(* PLC project Generated.project, CODESYS CODESYS V3.5 SP19 Patch 1 *)
(* stored: creationDateTime 2026-11-16T13:11:40.466311, modificationDateTime 2026-11-16T13:11:40.466311 *)

(* DOC: DOC/AF/AF_Partie-13_Fonction_Simulation_v2.5.md Capteur de position cumulatif avec hysteresis et episode intermittent rejouable. Cette brique ne connait ni le mouvement ni la logique M3 : elle transforme uniquement une position mecanique vraie en DI. *)
FUNCTION_BLOCK FB_Sim_PositionSensor
  VAR_INPUT
    Enable : BOOL;
    Position_M : REAL;
    Threshold_M : REAL;
    Hysteresis_M : REAL := 0.02;
    ActiveBelowThreshold : BOOL := TRUE;
    ElectricalDelayS : REAL := 0;
    IntermittenceActive : BOOL := FALSE;
    IntermittenceDurationS : REAL := 1;
    IntermittencePeriodS : REAL := 0.12;
    ScenarioSeed : UDINT := 1;
    CycleTimeS : REAL := 0.01;
    BlipTransitions : UDINT := 0;  (* Profil « BLIP COURT » — SECOND profil, independant du train de bascules du profil d'intermittence ci-dessus (dont les parametres restent inchanges). 0 = desactive : le comportement historique est strictement conserve. Rejoue les excursions electriques courtes mesurees sur la trace terrain du 2026-09-04 : Tremie contradictoire pendant 2 echantillons a 12,24 s (~200 ms) et PV reactive 1 echantillon a 14,94 s (~100 ms). BlipTransitions = nombre de bascules electriques (1 = une excursion puis retour) ; BlipDurationS = duree de maintien de chaque etat, donc largeur de l'excursion. *)
    BlipDurationS : REAL := 0.2;
    CamDropoutActive : BOOL := FALSE;  (* L5 (2026-10-28) — MECANISME DE CAME, SPATIAL : en franchissant le capteur on le VOIT, on le PERD sur une courte zone, on le RETROUVE, puis il reste FIXE. Lie a la POSITION (pas au temps) : se produit a chaque passage, dans les DEUX sens, et reste stable a l'arret (bornes de la zone avec hysteresis CST_CamHysteresis_M contre le bruit/balancement). Zone de perte placee APRES le front de detection (cote -/+ Hysteresis_M) : [front - Start - Width ; front - Start] cote detection. FALSE = historique strictement inchange. Valeurs = HYPOTHESES. *)
    CamDropoutStart_M : REAL := 0.02;
    CamDropoutWidth_M : REAL := 0.04;
    FiniteCamActive : BOOL := FALSE;  (* Came finie : FALSE = capteur cumulatif ; TRUE = sortie active uniquement sur CamLength_M apres Threshold_M. *)
    CamLength_M : REAL := 0;
  END_VAR
  VAR_OUTPUT
    RawDetected : BOOL;
    ElectricalOutput : BOOL;
    EpisodeActive : BOOL;
    BlipActive : BOOL;
    TransitionCount : UDINT;
    EpisodeTogglePeriodS : REAL;
  END_VAR
  VAR
    Initialized : BOOL;
    PreviousRawDetected : BOOL;
    EpisodeTarget : BOOL;
    DelayTimerS : REAL;
    EpisodeTimerS : REAL;
    ToggleTimerS : REAL;
    RandomState : UDINT;
    BlipRunning : BOOL;
    BlipTimerS : REAL;
    BlipCount : UDINT;
    HystDetected : BOOL;  (* L5 : etat mecanique avec hysteresis (avant perte de came) *)
    InCamDropout : BOOL;  (* L5 : position dans la zone de perte de la came *)
    CamNear_M : REAL;  (* L5 : borne de la zone cote front de detection *)
    CamFar_M : REAL;  (* L5 : borne de la zone cote interieur *)
    PastFiniteCam : BOOL;  (* Depassement au-dela de la longueur physique de came *)
    CamEnd_M : REAL;  (* Borne de fin de came finie *)
    CST_BlipMaxTransitions : UDINT := 1000;  (* Plafond du nombre de bascules du profil « blip court » : borne la duree de l'episode et interdit tout rebouclage de compteur UDINT (revue du 2026-09-20, F9). *)
    CST_CamHysteresis_M : REAL := 0.01;  (* L5 : hysteresis des bornes de la zone de perte *)
  END_VAR

            

IF NOT Enable THEN
    Initialized := FALSE;
    RawDetected := FALSE;
    ElectricalOutput := FALSE;
    PreviousRawDetected := FALSE;
    EpisodeActive := FALSE;
    BlipActive := FALSE;
    BlipRunning := FALSE;
    BlipTimerS := 0.0;
    BlipCount := 0;
    DelayTimerS := 0.0;
    EpisodeTimerS := 0.0;
    ToggleTimerS := 0.0;
    TransitionCount := 0;
    EpisodeTogglePeriodS := 0.0;
    PastFiniteCam := FALSE;
    RETURN;
END_IF;

(* Hysteresis sur une frontiere cumulative : les cinq DI restent compatibles avec
   le mot thermometre du decodeur M3, contrairement a cinq fenetres independantes. *)
IF NOT Initialized THEN
    IF ActiveBelowThreshold THEN
        RawDetected := Position_M <= Threshold_M;
        IF FiniteCamActive THEN
            PastFiniteCam := Position_M < (Threshold_M - MAX(0.0, CamLength_M));
            RawDetected := RawDetected AND NOT PastFiniteCam;
        ELSE
            PastFiniteCam := FALSE;
        END_IF;
    ELSE
        RawDetected := Position_M >= Threshold_M;
        IF FiniteCamActive THEN
            PastFiniteCam := Position_M > (Threshold_M + MAX(0.0, CamLength_M));
            RawDetected := RawDetected AND NOT PastFiniteCam;
        ELSE
            PastFiniteCam := FALSE;
        END_IF;
    END_IF;
    HystDetected := RawDetected;
    ElectricalOutput := RawDetected;
    PreviousRawDetected := RawDetected;
    RandomState := ScenarioSeed MOD 1000000;
    IF RandomState = 0 THEN
        RandomState := 1;
    END_IF;
    EpisodeTogglePeriodS := MAX(0.01, IntermittencePeriodS);
    Initialized := TRUE;
    RETURN;
END_IF;

IF ActiveBelowThreshold THEN
    IF HystDetected THEN
        HystDetected := Position_M <= (Threshold_M + MAX(0.0, Hysteresis_M));
    ELSE
        HystDetected := Position_M <= (Threshold_M - MAX(0.0, Hysteresis_M));
    END_IF;
    (* Zone de perte : apres le front d'entree en detection (cote - hysteresis), vers l'interieur. *)
    CamNear_M := Threshold_M - MAX(0.0, Hysteresis_M) - MAX(0.0, CamDropoutStart_M);
    CamFar_M := CamNear_M - MAX(0.0, CamDropoutWidth_M);
    IF NOT CamDropoutActive THEN
        InCamDropout := FALSE;
    ELSIF InCamDropout THEN
        InCamDropout := (Position_M <= CamNear_M + CST_CamHysteresis_M) AND (Position_M > CamFar_M - CST_CamHysteresis_M);
    ELSE
        InCamDropout := (Position_M <= CamNear_M - CST_CamHysteresis_M) AND (Position_M > CamFar_M + CST_CamHysteresis_M);
    END_IF;
    CamEnd_M := Threshold_M - MAX(0.0, CamLength_M);
    IF NOT FiniteCamActive THEN
        PastFiniteCam := FALSE;
    ELSIF PastFiniteCam THEN
        PastFiniteCam := Position_M < (CamEnd_M + CST_CamHysteresis_M);
    ELSE
        PastFiniteCam := Position_M < CamEnd_M;
    END_IF;
ELSE
    IF HystDetected THEN
        HystDetected := Position_M >= (Threshold_M - MAX(0.0, Hysteresis_M));
    ELSE
        HystDetected := Position_M >= (Threshold_M + MAX(0.0, Hysteresis_M));
    END_IF;
    CamNear_M := Threshold_M + MAX(0.0, Hysteresis_M) + MAX(0.0, CamDropoutStart_M);
    CamFar_M := CamNear_M + MAX(0.0, CamDropoutWidth_M);
    IF NOT CamDropoutActive THEN
        InCamDropout := FALSE;
    ELSIF InCamDropout THEN
        InCamDropout := (Position_M >= CamNear_M - CST_CamHysteresis_M) AND (Position_M < CamFar_M + CST_CamHysteresis_M);
    ELSE
        InCamDropout := (Position_M >= CamNear_M + CST_CamHysteresis_M) AND (Position_M < CamFar_M - CST_CamHysteresis_M);
    END_IF;
    CamEnd_M := Threshold_M + MAX(0.0, CamLength_M);
    IF NOT FiniteCamActive THEN
        PastFiniteCam := FALSE;
    ELSIF PastFiniteCam THEN
        PastFiniteCam := Position_M > (CamEnd_M - CST_CamHysteresis_M);
    ELSE
        PastFiniteCam := Position_M > CamEnd_M;
    END_IF;
END_IF;
(* L5 : perte de came + came finie ; hors options, RawDetected = HystDetected. *)
RawDetected := HystDetected AND NOT InCamDropout AND NOT PastFiniteCam;

(* Un episode est declenche par un franchissement mecanique, pas par une de ses
   propres bascules electriques. Les fronts restent donc bornes et reproductibles. *)
IF RawDetected <> PreviousRawDetected THEN
    PreviousRawDetected := RawDetected;
    EpisodeTarget := RawDetected;
    (* Une bascule mecanique pendant l'episode modifie seulement la cible finale.
       Elle ne remet jamais son chronometre a zero : l'episode reste borne. *)
    IF NOT EpisodeActive THEN
        DelayTimerS := 0.0;
        EpisodeTimerS := 0.0;
        ToggleTimerS := 0.0;
        (* Tirage unique par episode : reproductible pour une graine et sans bruit
           blanc scan-par-scan. La periode varie de 70 % a 130 % du nominal. *)
        RandomState := RandomState + 7919;
        IF RandomState >= 1000000 THEN
            RandomState := RandomState - 1000000;
        END_IF;
        EpisodeTogglePeriodS := MAX(0.01, IntermittencePeriodS
            * (0.7 + UDINT_TO_REAL(RandomState MOD 6000) / 10000.0));
        EpisodeActive := IntermittenceActive AND (IntermittenceDurationS > 0.0);
    END_IF;
    (* Blip court : arme sur le meme front MECANIQUE. Ses propres bascules electriques ne
       peuvent donc jamais le rearmer — meme protection que l'episode d'intermittence. *)
    IF (BlipTransitions > 0) AND (BlipDurationS > 0.0) THEN
        BlipRunning := TRUE;
        BlipTimerS := 0.0;
        BlipCount := 0;
        BlipActive := TRUE;
        (* Ecretage : au-dela de ce plafond, un compteur UDINT pourrait reboucler et rendre
           le blip non terminant (revue du 2026-09-20, F9). *)
        BlipTransitions := MIN(BlipTransitions, CST_BlipMaxTransitions);
    END_IF;
END_IF;

IF BlipRunning THEN
    (* Protocole du blip court : (0) la sortie rejoint d'abord l'etat MECANIQUE — le
       comportement nominal reste donc visible ; puis une excursion contradictoire toutes
       les BlipDurationS, donc de largeur BlipDurationS ; enfin la sortie est rendue a
       l'etat mecanique. Nombre d'excursions = BlipTransitions. *)
    BlipTimerS := BlipTimerS + CycleTimeS;
    IF BlipTimerS >= MAX(CycleTimeS, BlipDurationS) THEN
        BlipTimerS := 0.0;
        IF BlipCount = 0 THEN
            IF ElectricalOutput <> RawDetected THEN
                ElectricalOutput := RawDetected;
                TransitionCount := TransitionCount + 1;
            END_IF;
            BlipCount := 1;
        ELSIF BlipCount <= BlipTransitions THEN
            ElectricalOutput := NOT ElectricalOutput;
            TransitionCount := TransitionCount + 1;
            BlipCount := BlipCount + 1;
        ELSE
            BlipRunning := FALSE;
            BlipActive := FALSE;
            IF ElectricalOutput <> RawDetected THEN
                ElectricalOutput := RawDetected;
                TransitionCount := TransitionCount + 1;
            END_IF;
            DelayTimerS := 0.0;
        END_IF;
    END_IF;
ELSIF EpisodeActive THEN
    EpisodeTimerS := EpisodeTimerS + CycleTimeS;
    ToggleTimerS := ToggleTimerS + CycleTimeS;
    IF ToggleTimerS >= EpisodeTogglePeriodS THEN
        ElectricalOutput := NOT ElectricalOutput;
        ToggleTimerS := 0.0;
        TransitionCount := TransitionCount + 1;
    END_IF;
    IF EpisodeTimerS >= IntermittenceDurationS THEN
        EpisodeActive := FALSE;
        IF ElectricalOutput <> EpisodeTarget THEN
            ElectricalOutput := EpisodeTarget;
            TransitionCount := TransitionCount + 1;
        END_IF;
        DelayTimerS := 0.0;
    END_IF;
ELSIF ElectricalOutput <> RawDetected THEN
    DelayTimerS := DelayTimerS + CycleTimeS;
    IF DelayTimerS >= MAX(0.0, ElectricalDelayS) THEN
        ElectricalOutput := RawDetected;
        DelayTimerS := 0.0;
        TransitionCount := TransitionCount + 1;
    END_IF;
ELSE
    DelayTimerS := 0.0;
END_IF;

          
END_FUNCTION_BLOCK
